_w1 := Burkert_OSCAT_BASIC.SCALE_R(X := Config.HLT.Assets.Level.EU, I_LO := 0.0, I_HI := Config.HLT.Assets.Level.Analog_Scale.Eu_Max, O_LO := 0, O_HI := 100);
Config.HLT.Current_Level_PCT := _w1;
Config.HLT.Current_Temp := Config.HLT.Assets.Temperature.EU;
_w2 := True;
IF _w2 THEN
    HLT_Task_Manager_0(Config := Config); // HLT_Task_Manager
END_IF
Service_Water_0(SFCReset := Config.HLT.Service_Water_Destination.eTarget <> Service_Water_0.Current_Destination, Config := Config); // Service_Water
IF Config.HLT.Mode.eMode=eHLT_Modes.Off THEN _w3 := False; END_IF
Config.HLT.AutoFill.Brew_Active := _w3;
_w4 := True;
IF _w4 THEN
    Alarm_Manager_0(Config := Config); // Alarm_Manager
END_IF
_w5 := _w4;
IF _w5 THEN
    HLT_Valve_Manager_0(Config := Config); // HLT_Valve_Manager
END_IF
_w6 := _w5;
IF _w6 THEN
    HLT_PID_Manager_0(Config := Config); // HLT_PID_MANAGER
END_IF
_w7 := _w6;
IF _w7 THEN
    HLT_Status_Manager_0(Config := Config); // HLT_STATUS_MANAGER
END_IF
IF _w7 THEN
    HLT_VFD_Ctrl_0(Config := Config); // HLT_VFD_Ctrl
END_IF
R_TRIG_1(CLK := Config.HLT.Mode.eMode<>HLT_Tasks_0.Current_Mode); // R_trig
IF _w2 THEN
    HLT_Tasks_0(SFCReset := R_TRIG_1.Q, Config := Config); // HLT_Tasks
END_IF
Config.HLT.Assets.Level.Burkert.cAlarm_Config := Config.HLT.AutoFill.Current_Profile.Level;
Config.HLT.Assets.Temperature.Burkert.cAlarm_Config := Config.HLT.AutoFill.Current_Profile.Temperature;
Config.HLT.Assets.HTX_Inlet_TT.Burkert.cAlarm_Config := Config.HLT.AutoFill.Current_Profile.Temperature;
Config.HLT.Assets.HTX_Outlet_TT.Burkert.cAlarm_Config := Config.HLT.AutoFill.Current_Profile.Temperature;
_w8 := DaySeconds(Hour := Config.HLT.Profile[1].Enable_Hour, Minute := Config.HLT.Profile[1].Enable_Minute, Second := 0);
_w9 := DaySeconds(Hour := Config.HLT.Profile[2].Enable_Hour, Minute := Config.HLT.Profile[2].Enable_Minute, Second := 0);
_w10 := DaySeconds(Hour := Config.HLT.Profile[3].Enable_Hour, Minute := Config.HLT.Profile[3].Enable_Minute, Second := 0);
_w11 := DaySeconds(Hour := Config.HLT.Profile[4].Enable_Hour, Minute := Config.HLT.Profile[4].Enable_Minute, Second := 0);
_w12 := Burkert_OSCAT_BASIC.BIT_OF_DWORD(in := Config.HLT.Profile[0].Enable_Days, N := RTC.wDayOfWeek);
_w13 := DaySeconds(Hour := Config.HLT.Profile[0].Enable_Hour, Minute := Config.HLT.Profile[0].Enable_Minute, Second := 0);
_w14 := (_w12 AND Day_Seconds = _w13 OR Config.HLT.AutoFill.Brew_Active) AND (Config	.HLT.Mode.eMode=eHLT_Modes.Auto) OR (Config.HLT.Manual_Profile=0);
_w15 := Burkert_OSCAT_BASIC.BIT_OF_DWORD(in := Config.HLT.Profile[1].Enable_Days, N := RTC.wDayOfWeek);
_w16 := _w15 AND Day_Seconds = _w8 AND (Config	.HLT.Mode.eMode=eHLT_Modes.Auto) OR (Config.HLT.Manual_Profile=1);
_w17 := Burkert_OSCAT_BASIC.BIT_OF_DWORD(in := Config.HLT.Profile[2].Enable_Days, N := RTC.wDayOfWeek);
_w18 := _w17 AND Day_Seconds = _w9 AND (Config	.HLT.Mode.eMode=eHLT_Modes.Auto) OR (Config.HLT.Manual_Profile=2);
_w19 := Burkert_OSCAT_BASIC.BIT_OF_DWORD(in := Config.HLT.Profile[3].Enable_Days, N := RTC.wDayOfWeek);
_w20 := _w19 AND Day_Seconds = _w10 OR (Config.HLT.Manual_Profile=3);
_w21 := Burkert_OSCAT_BASIC.BIT_OF_DWORD(in := Config.HLT.Profile[4].Enable_Days, N := RTC.wDayOfWeek);
_w22 := _w21 AND Day_Seconds = _w11 AND (Config	.HLT.Mode.eMode=eHLT_Modes.Auto) AND False OR (Config.HLT.Manual_Profile=4);
_w23 := _w14 OR _w16 OR _w18 OR _w20 OR _w22;
_w24 := SEL(_w14, SEL(_w16, SEL(_w18, SEL(_w20, SEL(_w22, 5, 4), 3), 2), 1), 0);
_w25 := _w23;
IF _w25 THEN _w26 := MUX(_w24, Config.HLT.Profile[0], Config.HLT.Profile[1], Config.HLT.Profile[2], Config.HLT.Profile[3], Config.HLT.Profile[4]); END_IF
Config.HLT.AutoFill.Current_Profile := _w26;
R_TRIG_2(CLK := _w25); // R_trig
IF R_TRIG_2.Q THEN _w27 := eHLT_Task.Fill; END_IF
Config.HLT.Task.eTask := _w27;
_w28 := _w23;
IF _w28 THEN _w29 := _w24; END_IF
Config.HLT.Active_Profile := _w29;
IF _w28 THEN _w30 := 255; END_IF
Config	.HLT.Manual_Profile := _w30;

END_PROGRAM

// HLT_Task_Manager
FUNCTION_BLOCK HLT_Task_Manager
VAR_INPUT
END_VAR
VAR_OUTPUT
END_VAR
VAR
END_VAR


VAR_INPUT
	Config: REFERENCE TO Config_DUT;
END_VAR
VAR // added by the converter: edge detectors and wires of the graphical bodies
    _w1 : BOOL;
END_VAR

_w1 := Config.HLT.AutoFill.Current_Profile.Temperature.Setpoints.Hi_warn - Config.HLT.AutoFill.Current_Profile.Temperature.Setpoints.Low_warn >= 2.0;
Config.HLT.Task.eTask := SEL(Config.HLT.Mode.eMode=eHlt_Modes.Auto, Config.HLT.Task.eTask, SEL(Config.HLT.Service_Water.OpenDestination, SEL(Config.HLT.Assets.Level.Status.eStatus=Burkert.eSensor_Status.Low_Low_Alarm, SEL(Config.HLT.Assets.Level.Status.eStatus=Burkert.eSensor_Status.Low_Warning, SEL(_w1 AND (Config.HLT.Assets.Temperature.EU < (Config.HLT.AutoFill.Current_Profile.Temperature.Setpoints.Low_warn+0.1)) OR (Config.HLT.Assets.Level.EU>(Config.HLT.Assets.Level.Burkert.cAlarm_Config.Hi_Warn-10)), SEL(_w1 AND (Config.HLT.Assets.Temperature.EU > (Config.HLT.AutoFill.Current_Profile.Temperature.Setpoints.Hi_warn-0.2)), SEL(NOT _w1 AND (Config.HLT.Assets.Temperature.EU > (Config.HLT.AutoFill.Current_Profile.Temperature.Setpoints.Low_warn)), Config.HLT.Task.eTask, eHLT_Task.Ready_Holding), eHLT_Task.Ready), eHLT_Task.Heat_Recirculate), eHLT_Task.Fill_Heat), eHLT_Task.Fill), eHLT_Task.Line_Chase));

END_FUNCTION_BLOCK

// Service_Water
FUNCTION_BLOCK Service_Water
VAR
	TransferLoop:Batch_Transfer;
	Current_Destination:INT;
	Current_Mode:INT;
	lclStatus:Transfer_Status;
END_VAR

VAR_INPUT
	SFCReset:BOOL;
	//Config.HLT.Service_Water.DestinationOpen:BOOL;
END_VAR

VAR_OUTPUT
	SFCcurrentStep:STRING[49];
	//Config.HLT.Service_Water.OpenDestination:BOOL;
END_VAR

VAR_IN_OUT
	//transfer:cBatch_Transfer;
END_VAR
VAR_INPUT
	Config: REFERENCE TO Config_DUT;
END_VAR

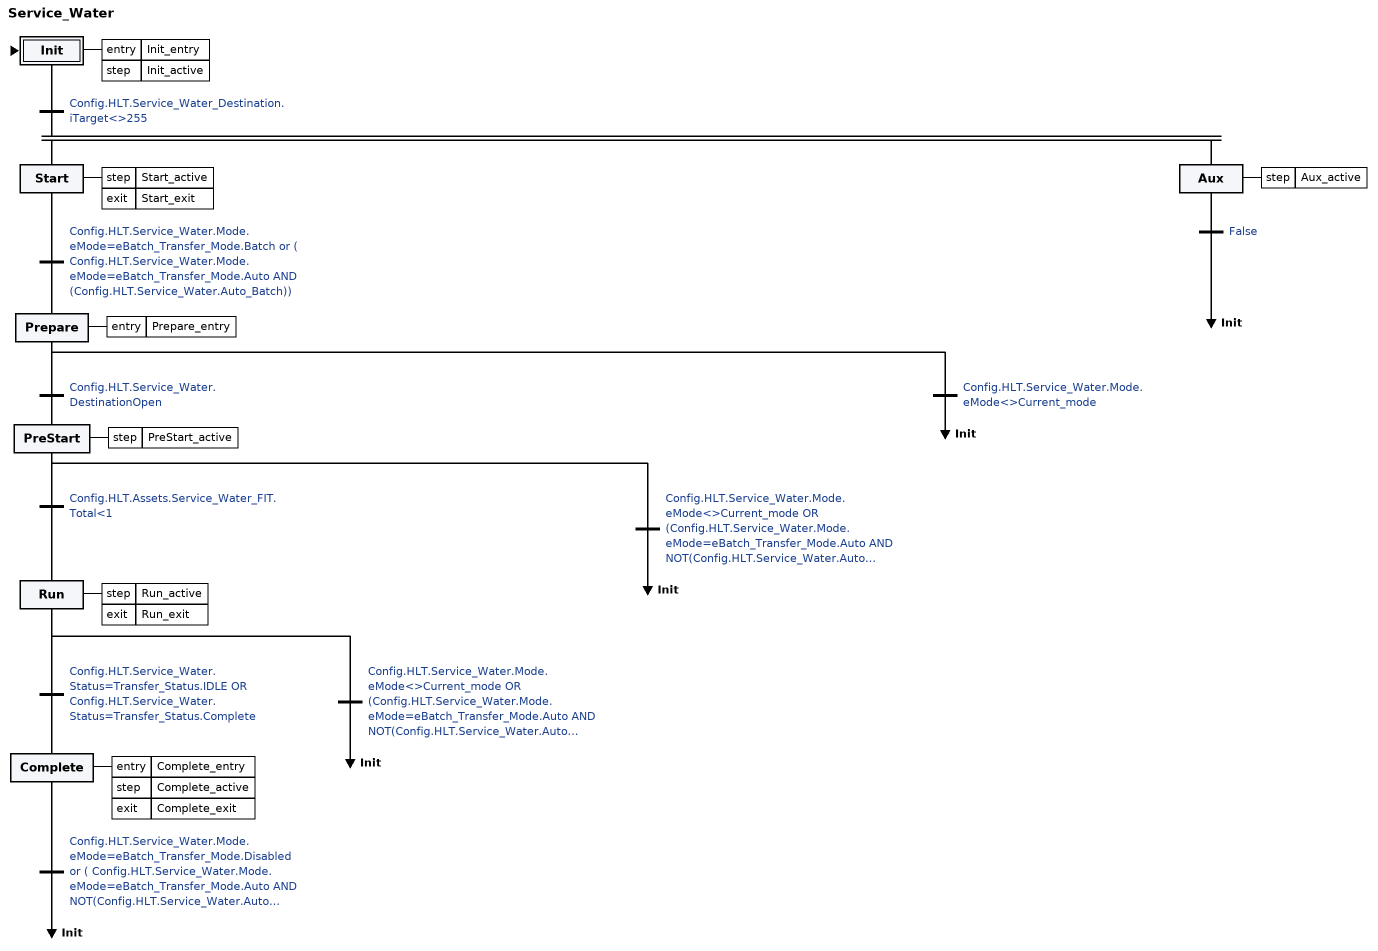
INITIAL_STEP Init:
    Init_entry(P1);  // entry action
    Init_active(N);  // step action
END_STEP
TRANSITION FROM Init TO (Start, Aux)
    := Config.HLT.Service_Water_Destination.iTarget<>255;
END_TRANSITION
STEP Start:
    Start_active(N);  // step action
    Start_exit(P0);  // exit action
END_STEP
STEP Aux:
    Aux_active(N);  // step action
END_STEP
TRANSITION FROM Aux TO Init
    := False;
END_TRANSITION
TRANSITION FROM Start TO Prepare
    := Config.HLT.Service_Water.Mode.eMode=eBatch_Transfer_Mode.Batch or ( Config.HLT.Service_Water.Mode.eMode=eBatch_Transfer_Mode.Auto AND (Config.HLT.Service_Water.Auto_Batch));
END_TRANSITION
STEP Prepare:
    Prepare_entry(P1);  // entry action
END_STEP
TRANSITION FROM Prepare TO PreStart
    := Config.HLT.Service_Water.DestinationOpen;
END_TRANSITION
TRANSITION FROM Prepare TO Init
    := Config.HLT.Service_Water.Mode.eMode<>Current_mode;
END_TRANSITION
STEP PreStart:
    PreStart_active(N);  // step action
END_STEP
TRANSITION FROM PreStart TO Run
    := Config.HLT.Assets.Service_Water_FIT.Total<1;
END_TRANSITION
TRANSITION FROM PreStart TO Init
    := Config.HLT.Service_Water.Mode.eMode<>Current_mode OR (Config.HLT.Service_Water.Mode.eMode=eBatch_Transfer_Mode.Auto AND NOT(Config.HLT.Service_Water.Auto_Batch));
END_TRANSITION
STEP Run:
    Run_active(N);  // step action
    Run_exit(P0);  // exit action
END_STEP
TRANSITION FROM Run TO Complete
    := Config.HLT.Service_Water.Status=Transfer_Status.IDLE OR Config.HLT.Service_Water.Status=Transfer_Status.Complete;
END_TRANSITION
TRANSITION FROM Run TO Init
    := Config.HLT.Service_Water.Mode.eMode<>Current_mode OR (Config.HLT.Service_Water.Mode.eMode=eBatch_Transfer_Mode.Auto AND NOT(Config.HLT.Service_Water.Auto_Batch));
END_TRANSITION
STEP Complete:
    Complete_entry(P1);  // entry action
    Complete_active(N);  // step action
    Complete_exit(P0);  // exit action
END_STEP
TRANSITION FROM Complete TO Init
    := Config.HLT.Service_Water.Mode.eMode=eBatch_Transfer_Mode.Disabled or ( Config.HLT.Service_Water.Mode.eMode=eBatch_Transfer_Mode.Auto AND NOT(Config.HLT.Service_Water.Auto_Batch));
END_TRANSITION

END_FUNCTION_BLOCK

// HLT_VFD_Ctrl
FUNCTION_BLOCK HLT_VFD_Ctrl
VAR
END_VAR
VAR_INPUT
	Config: REFERENCE TO Config_DUT;
END_VAR
VAR // added by the converter: edge detectors and wires of the graphical bodies
    _w1, _w2 : ANY;
END_VAR

_w1 := (Config.HLT.Assets.SprayBall.Status=Burkert.eBCV_Status.A_Open) AND (Config.HLT.Task.eTask=eHLT_Task.Spray_Ball);
Config.HLT.Assets.Mix_Pump.PLC_Run := (Config.HLT.Assets.Strike_HW.Valve_Actual>5) OR (Config.HLT.Assets.Sparge_HW.Valve_Actual>5) OR _w1;
Config.HLT.Assets.Mix_Pump.PLC_CMD := SEl(_w1, MAX(Config.HLT.Assets.Sparge_HW.Valve_Actual, Config.HLT.Assets.Strike_HW.Valve_Actual), Config.HLT.Spray_Ball_Rate);
_w2 := Config.HLT.Assets.PID_Recirc.CV + (Config	.HLT.Service_Water.ACV);
Config.HLT.Assets.Recirc_Pump.PLC_CMD := SEL(_w2 <= 15, LIMIT(0.0, 100.0, _w2), 15);
Config.HLT.Assets.Recirc_Pump.PLC_Run := 5 < _w2;
// Config.HLT.Assets.Sparge_CW.Valve_Actual>5: input not connected
// Config.HLT.Assets.Strike_HW.Valve_Actual>5: input not connected
// Config.HLT.Assets.PID_Recirc.CV>2: input not connected

END_FUNCTION_BLOCK

// HLT_Valve_Manager
FUNCTION_BLOCK HLT_Valve_Manager
VAR
	//TOF_0: TOF;
END_VAR
VAR_INPUT
	Config: REFERENCE TO Config_DUT;
END_VAR
VAR // added by the converter: edge detectors and wires of the graphical bodies
    _w1, _w2 : ANY;
END_VAR

_w1 := (Config.HLT.Task.eTask=eHLT_Task.Heat_Recirculate) OR (Config.HLT.Task.eTask=eHLT_Task.Fill) OR (Config.HLT.Task.eTask=eHLT_Task.Fill_Heat) OR (Config.HLT.Task.eTask=eHLT_Task.Ready) OR (Config.HLT.Task.eTask=eHLT_Task.Spray_Ball);
Config.HLT.Assets.HTX_Steam.PLC_CMD := MAX(Config.HLT.Assets.PID_HTX.CV, 0.0);
_w2 := NOT (Config.HLT.Mode.eMode=eHLT_Modes.Off) AND Config.HLT.Assets.Level.Ready AND (Config.HLT.Assets.Level.Status.eStatus<>Burkert.eSensor_Status.HiHi_Alarm) AND ((Config.HLT.Task.eTask=eHLT_Task.Fill) OR (Config.HLT.Task.eTask=eHLT_Task.Fill_Heat));
Config.HLT.Assets.CW_Fill.PLC_CMD := _w2;
Config.HLT.Assets.Recirc_To_HTX.PLC_CMD := _w1;
Config.HLT.Assets.HTX_Outlet_ACV.PLC_CMD := SEL(Config.HLT.Task.eTask=eHLT_Task.Line_Chase, SEL(_w2, SEL((Config.HLT.Task.eTask=eHLT_Task.Ready_Holding) OR (Config.HLT.Task.eTask=eHLT_Task.Heat_Recirculate) OR (Config.HLT.Task.eTask=eHLT_Task.Ready) OR Config.HLT.Assets.PID_Recirc.PLC_Enable, 0.0, Config.HLT.Assets.PID_Recirc.CV), 100), Config.HLT.Assets.PID_Recirc.CV);
Config.HLT.Assets.SprayBall.PLC_CMD := (Config.HLT.Task.eTask=eHLT_Task.Spray_Ball) OR False;

END_FUNCTION_BLOCK

// HLT_PID_Manager
FUNCTION_BLOCK HLT_PID_Manager
VAR 
	RAMP_REAL_0: RAMP_REAL;
END_VAR
VAR_INPUT
	Config: REFERENCE TO Config_DUT;
END_VAR


//Config.HLT.Assets.HTX_FIT
VAR // added by the converter: edge detectors and wires of the graphical bodies
    _w1, _w2, _w4 : BOOL;
    _w3, _w5 : ANY;
END_VAR

Config.HLT.Assets.PID_HTX.Actual := Config.HLT.Assets.HTX_Outlet_TT.EU;
Config.HLT.Assets.PID_Recirc.Actual := Config.HLT.Assets.HTX_FIT.Rate;
_w1 := (Config.HLT.Task.eTask=eHLT_Task.Line_Chase) OR (Config.HLT.Task.eTask=eHLT_Task.Heat_Recirculate) OR (Config.HLT.Task.eTask=eHLT_Task.Ready_Holding) OR False;
_w2 := ((Config.HLT.Task.eTask=eHLT_Task.Line_Chase) OR (Config.HLT.Task.eTask=eHLT_Task.Heat_Recirculate) OR (Config.HLT.Task.eTask=eHLT_Task.Ready_Holding) OR False OR (Config.HLT.Task.eTask=eHLT_Task.Heat_Recirculate) OR (Config.HLT.Task.eTask=eHLT_Task.Fill_Heat)) AND (Config.HLT.Assets.HTX_FIT.Rate>10);
IF _w2 THEN _w3 := SEL(Config.HLT.Task.eTask=eHLT_Task.Ready_Holding, Config.HLT.AutoFill.Current_Profile.Temperature.Setpoints.Hi_warn, Config.HLT.AutoFill.Current_Profile.Temperature.Setpoints.Low_warn + (Config.HLT.AutoFill.Current_Profile.Temperature.Setpoints.Hi_warn - Config.HLT.AutoFill.Current_Profile.Temperature.Setpoints.Low_warn) / 2.0); END_IF
Config.HLT.Assets.PID_HTX.PLC_Target := _w3;
Config.HLT.Assets.PID_HTX.PLC_Enable := _w2;
RAMP_REAL_0(
    IN := SEL(Config.HLT.Assets.PID_Recirc.CV>99, Config.HLT.recirc_Rate + Config.HLT.Service_Water.Config.Rate, Config.HLT.Service_Water.Config.Rate),
    ASCEND := 5,
    DESCEND := 1,
    TIMEBASE := T#2s,
    RESET := False); // RAMP_REAL
_w4 := _w1;
IF _w4 THEN _w5 := SEL(Config.HLT.Task.eTask=eHLT_Task.Line_Chase, Config.HLT.recirc_Rate, RAMP_REAL_0.OUT); END_IF
Config.HLT.Assets.PID_Recirc.PLC_Target := _w5;
Config.HLT.Assets.PID_Recirc.PLC_Enable := _w4;

END_FUNCTION_BLOCK

// HLT_Status_Manager
FUNCTION_BLOCK HLT_Status_Manager
VAR
	TON_0: TON;
END_VAR
VAR_INPUT
	Config: REFERENCE TO Config_DUT;
END_VAR

//Config.HLT.Assets.CW_Fill

(* body of a kind this reader does not render *)

END_FUNCTION_BLOCK

// Service_Water_Manager
FUNCTION_BLOCK Service_Water_Manager
VAR
	//tStr_Destination:Service_Water_mapping;
	Service_Water_0: Service_Water;
END_VAR

VAR_INPUT
	Config: REFERENCE TO Config_DUT;
END_VAR
VAR // added by the converter: edge detectors and wires of the graphical bodies
    _w1, _w2, _w3, _w4, _w5, _w6, _w7 : ANY;
END_VAR

_w1 := (Config.HLT.Service_Water_Destination.eTarget=Service_Water_mapping.MLT_Vessel) AND (Config.MM.Status=eMM_Status.Rinse_Vessel);
_w2 := (Config.HLT.Service_Water_Destination.eTarget=Service_Water_mapping.KTWP_Sprayball) AND (Config.KT.Status=eKT_Status.Rinse);
_w3 := (Config.HLT.Service_Water_Destination.eTarget=Service_Water_mapping.Grant_Chase) AND (Config.MM.Status=eMM_Status.Rinse_Grant) AND (GVL.BCV[BCV_Mapping.BCV_008_Drain_BCV].Status=Burkert.eBCV_Status.A_Open) AND (GVL.BCV[BCV_Mapping.BCV_010_Grant_Out].Status=Burkert.eBCV_Status.A_Open);
_w4 := (Config.HLT.Service_Water_Destination.eTarget=Service_Water_mapping.KTWP_Low_Outlet) AND (Config.KT.Status=eKT_Status.Rinse_Low_Outlet);
_w5 := (Config.HLT.Service_Water_Destination.eTarget=Service_Water_mapping.CastOut_Chase) AND ((Config.KT.Status=eKT_Status.CastOut_Chase_Start) OR (Config.KT.Status=eKT_Status.CastOut_Chase_Active));
_w6 := (Config.HLT.Service_Water_Destination.eTarget=Service_Water_mapping.KTWP_Sprayball) AND (Config.KT.Status=eKT_Status.Rinse_Tank);
_w7 := (Config.HLT.Service_Water_Destination.eTarget=Service_Water_mapping.MLT_Transfer_Chase) AND ((Config.MM.Status=eMM_Status.Transfer_Chase_Ready) OR (Config.MM.Status=eMM_Status.Transfer_Chase_Active));
Config.HLT.Service_Water.DestinationOpen := MUX(Config	.HLT	.Service_Water_Destination.iTarget, GVL.BCV[BCV_Mapping.Underlet].Status=Burkert.eBCV_Status.A_Open, GVL.BCV[BCV_Mapping.BCV_028_MLT_Line_Chase].Status=Burkert.eBCV_Status.A_Open, GVL.BCV[BCV_Mapping.BCV_031_Grant_Spray_Ball].Status=Burkert.eBCV_Status.A_Open, GVL.BCV[BCV_Mapping.BCV_001_KTWP_Service_water_in].Status=Burkert.eBCV_Status.A_Open, GVL.BCV[BCV_Mapping.BCV_029_rinse_valve ].Status=Burkert.eBCV_Status.A_Open, (GVL.BCV[BCV_Mapping.KTWP_Spray_Ball].Status=Burkert.eBCV_Status.A_Open) AND (GVL.BCV[BCV_Mapping.BCV_039].Status=Burkert.eBCV_Status.A_Open) AND (GVL.BCV[BCV_Mapping.BCV_001_KTWP_Service_water_in].Status=Burkert.eBCV_Status.A_Open), (GVL.BCV[BCV_Mapping.BCV_017_KTWP_Tangent_Recirc].Status=Burkert.eBCV_Status.A_Open) AND (GVL.BCV[BCV_Mapping.BCV_039].Status=Burkert.eBCV_Status.A_Open) AND (GVL.BCV[BCV_Mapping.BCV_001_KTWP_Service_water_in].Status=Burkert.eBCV_Status.A_Open), (GVL.BCV[BCV_Mapping.BCV_001_KTWP_Service_water_in].Status=Burkert.eBCV_Status.A_Open) AND (GVL.BCV[BCV_Mapping.BCV_023_KTWP_High_outlet].Status=Burkert.eBCV_Status.A_Open), (GVL.BCV[BCV_Mapping.BCV_001_KTWP_Service_water_in].Status=Burkert.eBCV_Status.A_Open) AND (GVL.BCV[BCV_Mapping.BCV_024_KTWP_Low_Outlet].Status=Burkert.eBCV_Status.A_Open), False);
Config.HLT.Service_Water.Auto_Batch := (Config.HLT.Service_Water.Mode.eMode=eBatch_Transfer_Mode.Auto) AND ((Config.HLT.Service_Water_Destination.eTarget=Service_Water_mapping.CastOut_Chase) AND (Config.KT.Status=eKT_Status.CastOut_Chase_Active) OR (Config.HLT.Service_Water_Destination.eTarget=Service_Water_mapping.MLT_UnderLet) AND ((Config.MM.Status=eMM_Status.Underlet_Start) OR (Config.MM.Status=eMM_Status.Underlet_Active) OR (Config.MM.Status=eMM_Status.Rinse_Underlet)) OR _w7 OR _w5 OR _w3 OR _w1 OR _w2 OR (Config.HLT.Service_Water_Destination.eTarget=Service_Water_mapping.KTWP_High_Outlet) AND (Config.KT.Status=eKT_Status.Rinse_High_Outlet) OR _w6 OR _w4);

END_FUNCTION_BLOCK

// HLT_Tasks_OLD
FUNCTION_BLOCK HLT_Tasks_OLD
VAR
	Current_Task:eHLT_Task;
	Current_Mode:eHLT_Modes;
END_VAR

VAR_INPUT
	SFCReset:BOOL;
	
END_VAR

VAR_OUTPUT
	SFCcurrentStep:STRING[49];
END_VAR
VAR_INPUT
	Config: REFERENCE TO Config_DUT;
END_VAR

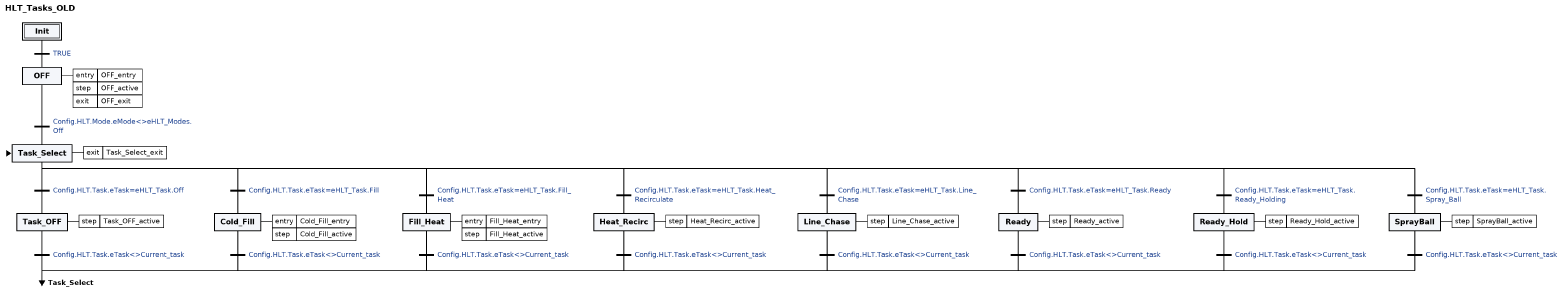
INITIAL_STEP Init:
END_STEP
TRANSITION FROM Init TO OFF
    := TRUE;
END_TRANSITION
STEP OFF:
    OFF_entry(P1);  // entry action
    OFF_active(N);  // step action
    OFF_exit(P0);  // exit action
END_STEP
TRANSITION FROM OFF TO Task_Select
    := Config.HLT.Mode.eMode<>eHLT_Modes.Off;
END_TRANSITION
STEP Task_Select:
    Task_Select_exit(P0);  // exit action
END_STEP
TRANSITION FROM Task_Select TO Task_OFF
    := Config.HLT.Task.eTask=eHLT_Task.Off;
END_TRANSITION
STEP Task_OFF:
    Task_OFF_active(N);  // step action
END_STEP
TRANSITION FROM Task_OFF TO Task_Select
    := Config.HLT.Task.eTask<>Current_task;
END_TRANSITION
TRANSITION FROM Task_Select TO Cold_Fill
    := Config.HLT.Task.eTask=eHLT_Task.Fill;
END_TRANSITION
STEP Cold_Fill:
    Cold_Fill_entry(P1);  // entry action
    Cold_Fill_active(N);  // step action
END_STEP
TRANSITION FROM Cold_Fill TO Task_Select
    := Config.HLT.Task.eTask<>Current_task;
END_TRANSITION
TRANSITION FROM Task_Select TO Fill_Heat
    := Config.HLT.Task.eTask=eHLT_Task.Fill_Heat;
END_TRANSITION
STEP Fill_Heat:
    Fill_Heat_entry(P1);  // entry action
    Fill_Heat_active(N);  // step action
END_STEP
TRANSITION FROM Fill_Heat TO Task_Select
    := Config.HLT.Task.eTask<>Current_task;
END_TRANSITION
TRANSITION FROM Task_Select TO Heat_Recirc
    := Config.HLT.Task.eTask=eHLT_Task.Heat_Recirculate;
END_TRANSITION
STEP Heat_Recirc:
    Heat_Recirc_active(N);  // step action
END_STEP
TRANSITION FROM Heat_Recirc TO Task_Select
    := Config.HLT.Task.eTask<>Current_task;
END_TRANSITION
TRANSITION FROM Task_Select TO Line_Chase
    := Config.HLT.Task.eTask=eHLT_Task.Line_Chase;
END_TRANSITION
STEP Line_Chase:
    Line_Chase_active(N);  // step action
END_STEP
TRANSITION FROM Line_Chase TO Task_Select
    := Config.HLT.Task.eTask<>Current_task;
END_TRANSITION
TRANSITION FROM Task_Select TO Ready
    := Config.HLT.Task.eTask=eHLT_Task.Ready;
END_TRANSITION
STEP Ready:
    Ready_active(N);  // step action
END_STEP
TRANSITION FROM Ready TO Task_Select
    := Config.HLT.Task.eTask<>Current_task;
END_TRANSITION
TRANSITION FROM Task_Select TO Ready_Hold
    := Config.HLT.Task.eTask=eHLT_Task.Ready_Holding;
END_TRANSITION
STEP Ready_Hold:
    Ready_Hold_active(N);  // step action
END_STEP
TRANSITION FROM Ready_Hold TO Task_Select
    := Config.HLT.Task.eTask<>Current_task;
END_TRANSITION
TRANSITION FROM Task_Select TO SprayBall
    := Config.HLT.Task.eTask=eHLT_Task.Spray_Ball;
END_TRANSITION
STEP SprayBall:
    SprayBall_active(N);  // step action
END_STEP
TRANSITION FROM SprayBall TO Task_Select
    := Config.HLT.Task.eTask<>Current_task;
END_TRANSITION

END_FUNCTION_BLOCK

// CIP_CTRL
PROGRAM CIP_CTRL
VAR
	R_TRIG_0: R_Trig;
	TON_0: TON;
	TON_1: TON;
	R_TRIG_1: R_Trig;
	TP_0: TP;
	TP_1: TP;
	TON_2: TON;
	Stage_Target_Out: REAL;
	Stage_Target_IN: REAL;
	TON_3: TON;
	F_TRIG_0: F_trig;
	Cip_Mode_tmp:eCIP_Modes;
	TP_2: TP;
	TP_3: TP;
	F_TRIG_1: F_trig;
	TON_4: TON;
	R_TRIG_2: R_trig;
	TP_4: TP;

	TON_3a: TON;
	TON_5: TON;
	TON_6: TON;
END_VAR
VAR // added by the converter: edge detectors and wires of the graphical bodies
    _w1, _w2, _w3, _w4, _w5, _w6, _w7, _w8, _w9, _w10, _w11, _w12, _w13, _w14, _w15, _w16, _w17, _w18, _w19, _w20, _w21, _w22, _w23 : BOOL;
    _rt1, _rt2, _rt3, _rt4, _rt5 : R_TRIG;
    _ft1 : F_TRIG;
END_VAR

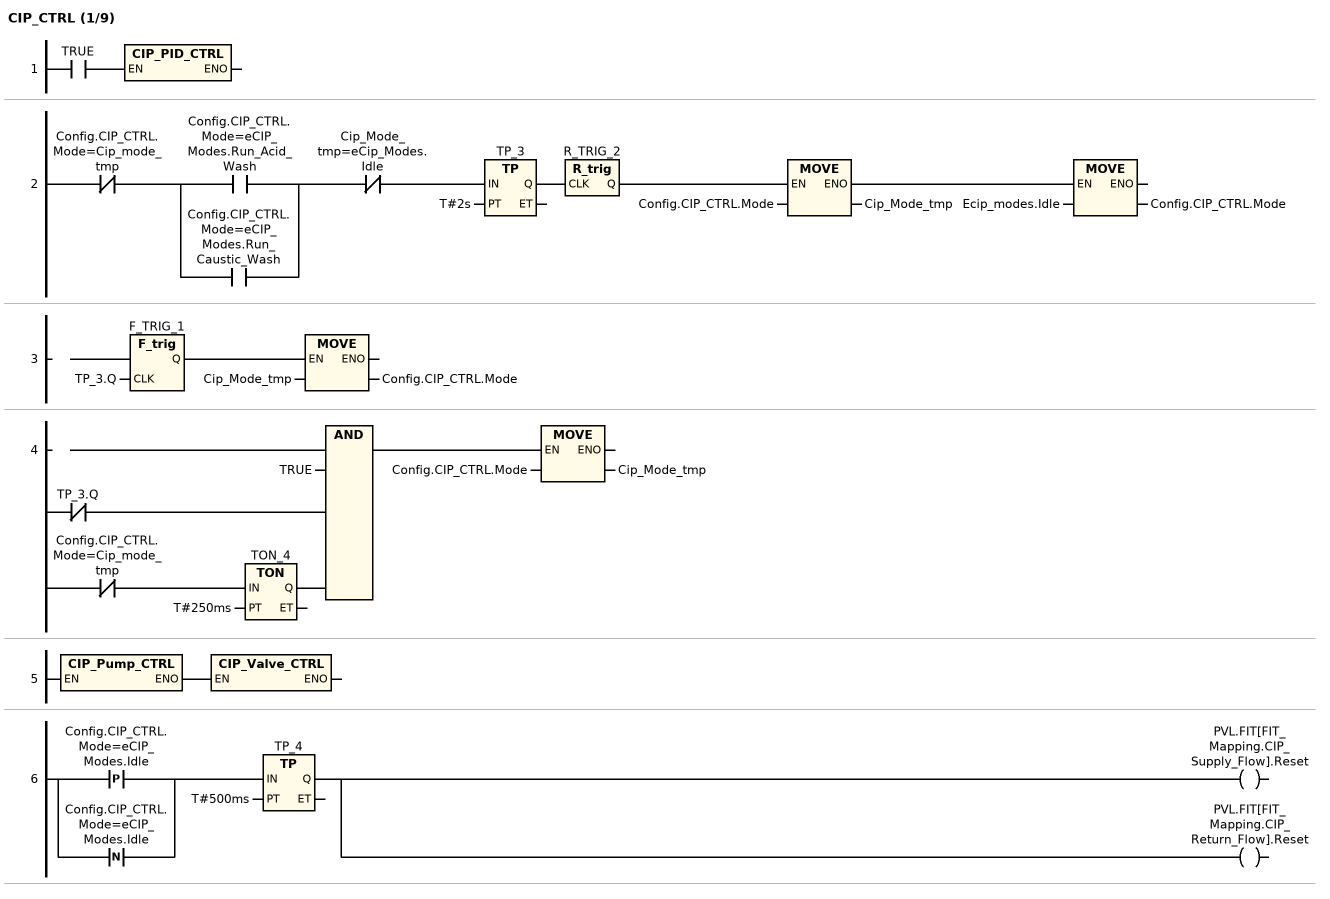
// NETWORK 1
CIP_PID_CTRL();

// NETWORK 2
TP_3(IN := NOT (Config.CIP_CTRL.Mode=Cip_mode_tmp) AND ((Config.CIP_CTRL.Mode=eCIP_Modes.Run_Acid_Wash) OR (Config.CIP_CTRL.Mode=eCIP_Modes.Run_Caustic_Wash)) AND NOT (Cip_Mode_tmp=eCip_Modes.Idle), PT := T#2s); // TP
R_TRIG_2(CLK := TP_3.Q); // R_trig
_w1 := R_TRIG_2.Q;
IF _w1 THEN Cip_Mode_tmp := Config.CIP_CTRL.Mode; END_IF
IF _w1 THEN Config.CIP_CTRL.Mode := Ecip_modes.Idle; END_IF

// NETWORK 3
F_TRIG_1(CLK := TP_3.Q); // F_trig
IF F_TRIG_1.Q THEN Config.CIP_CTRL.Mode := Cip_Mode_tmp; END_IF

// NETWORK 4
TON_4(IN := NOT (Config.CIP_CTRL.Mode=Cip_mode_tmp), PT := T#250ms); // TON
IF TRUE AND NOT TP_3.Q AND TON_4.Q THEN Cip_Mode_tmp := Config.CIP_CTRL.Mode; END_IF

// NETWORK 5
CIP_Pump_CTRL();
CIP_Valve_CTRL();

// NETWORK 6
_rt1(CLK := Config.CIP_CTRL.Mode=eCIP_Modes.Idle);
_ft1(CLK := Config.CIP_CTRL.Mode=eCIP_Modes.Idle);
TP_4(IN := _rt1.Q OR _ft1.Q, PT := T#500ms); // TP
PVL.FIT[FIT_Mapping.CIP_Supply_Flow].Reset := TP_4.Q;
PVL.FIT[FIT_Mapping.CIP_Return_Flow].Reset := TP_4.Q;

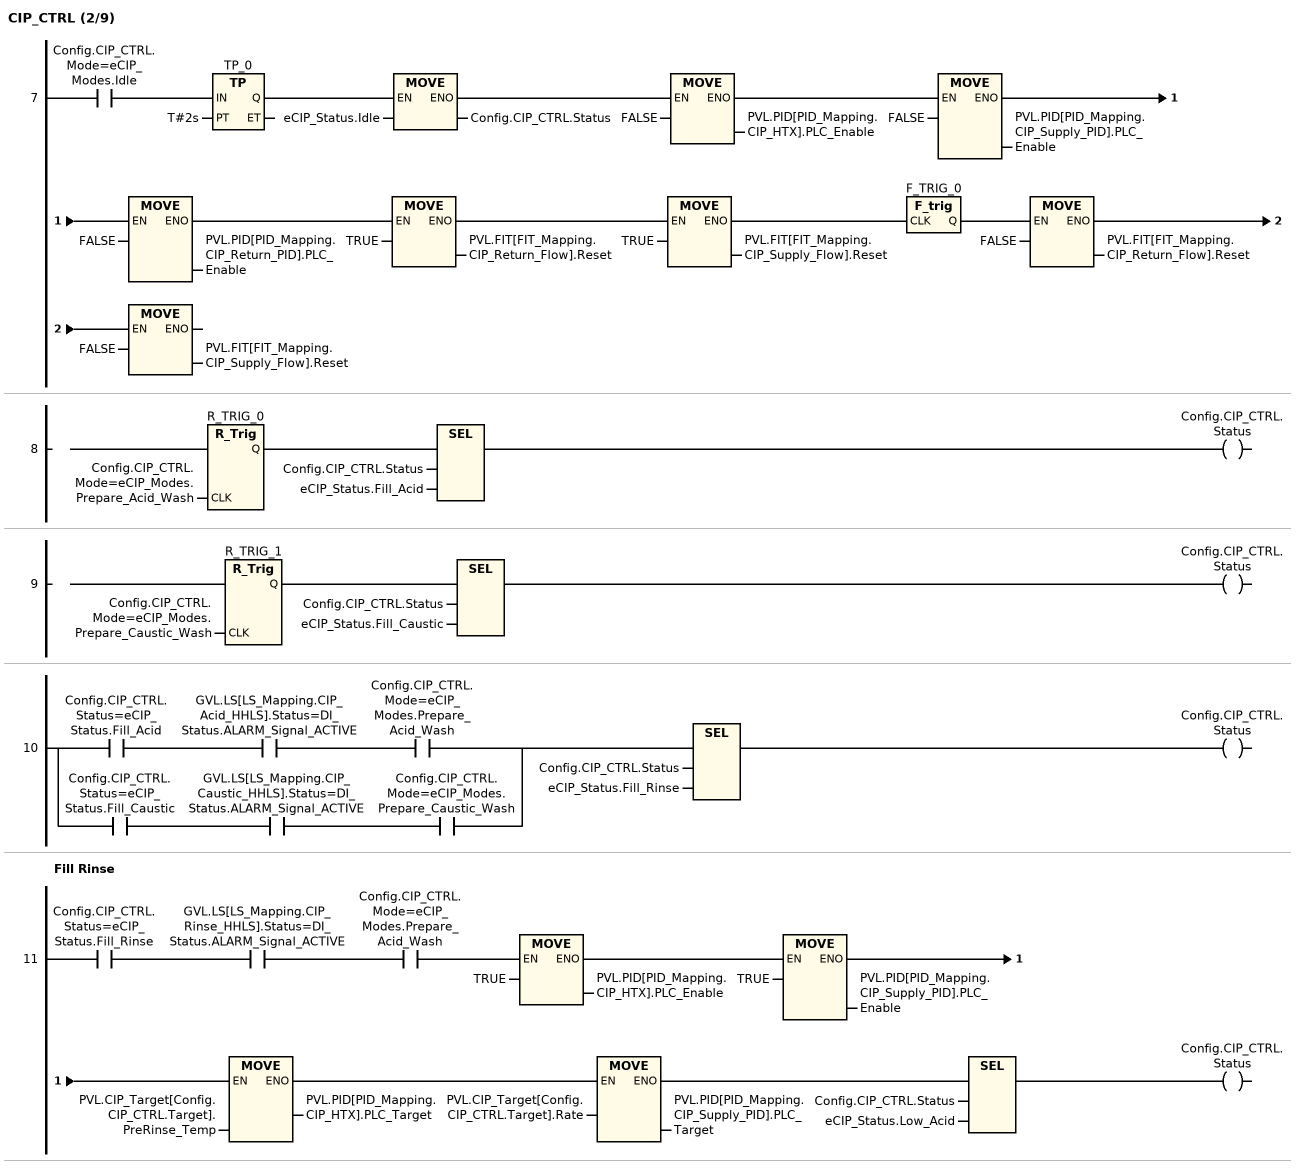
// NETWORK 7
TP_0(IN := Config.CIP_CTRL.Mode=eCIP_Modes.Idle, PT := T#2s); // TP
_w2 := TP_0.Q;
IF _w2 THEN Config.CIP_CTRL.Status := eCIP_Status.Idle; END_IF
IF _w2 THEN PVL.PID[PID_Mapping.CIP_HTX].PLC_Enable := FALSE; END_IF
IF _w2 THEN PVL.PID[PID_Mapping.CIP_Supply_PID].PLC_Enable := FALSE; END_IF
IF _w2 THEN PVL.PID[PID_Mapping.CIP_Return_PID].PLC_Enable := FALSE; END_IF
IF _w2 THEN PVL.FIT[FIT_Mapping.CIP_Return_Flow].Reset := TRUE; END_IF
IF _w2 THEN PVL.FIT[FIT_Mapping.CIP_Supply_Flow].Reset := TRUE; END_IF
F_TRIG_0(CLK := _w2); // F_trig
_w3 := F_TRIG_0.Q;
IF _w3 THEN PVL.FIT[FIT_Mapping.CIP_Return_Flow].Reset := FALSE; END_IF
IF _w3 THEN PVL.FIT[FIT_Mapping.CIP_Supply_Flow].Reset := FALSE; END_IF

// NETWORK 8
R_TRIG_0(CLK := Config.CIP_CTRL.Mode=eCIP_Modes.Prepare_Acid_Wash); // R_Trig
Config.CIP_CTRL.Status := SEL(R_TRIG_0.Q, Config.CIP_CTRL.Status, eCIP_Status.Fill_Acid);

// NETWORK 9
R_TRIG_1(CLK := Config.CIP_CTRL.Mode=eCIP_Modes.Prepare_Caustic_Wash); // R_Trig
Config.CIP_CTRL.Status := SEL(R_TRIG_1.Q, Config.CIP_CTRL.Status, eCIP_Status.Fill_Caustic);

// NETWORK 10
Config.CIP_CTRL.Status := SEL((Config.CIP_CTRL.Status=eCIP_Status.Fill_Acid) AND (GVL.LS[LS_Mapping.CIP_Acid_HHLS].Status=DI_Status.ALARM_Signal_ACTIVE) AND (Config.CIP_CTRL.Mode=eCIP_Modes.Prepare_Acid_Wash) OR (Config.CIP_CTRL.Status=eCIP_Status.Fill_Caustic) AND (GVL.LS[LS_Mapping.CIP_Caustic_HHLS].Status=DI_Status.ALARM_Signal_ACTIVE) AND (Config.CIP_CTRL.Mode=eCIP_Modes.Prepare_Caustic_Wash), Config.CIP_CTRL.Status, eCIP_Status.Fill_Rinse);

// NETWORK 11: Fill Rinse
_w4 := (Config.CIP_CTRL.Status=eCIP_Status.Fill_Rinse) AND (GVL.LS[LS_Mapping.CIP_Rinse_HHLS].Status=DI_Status.ALARM_Signal_ACTIVE) AND (Config.CIP_CTRL.Mode=eCIP_Modes.Prepare_Acid_Wash);
IF _w4 THEN PVL.PID[PID_Mapping.CIP_HTX].PLC_Enable := TRUE; END_IF
IF _w4 THEN PVL.PID[PID_Mapping.CIP_Supply_PID].PLC_Enable := TRUE; END_IF
IF _w4 THEN PVL.PID[PID_Mapping.CIP_HTX].PLC_Target := PVL.CIP_Target[Config.CIP_CTRL.Target].PreRinse_Temp; END_IF
IF _w4 THEN PVL.PID[PID_Mapping.CIP_Supply_PID].PLC_Target := PVL.CIP_Target[Config.CIP_CTRL.Target].Rate; END_IF
Config.CIP_CTRL.Status := SEL(_w4, Config.CIP_CTRL.Status, eCIP_Status.Low_Acid);

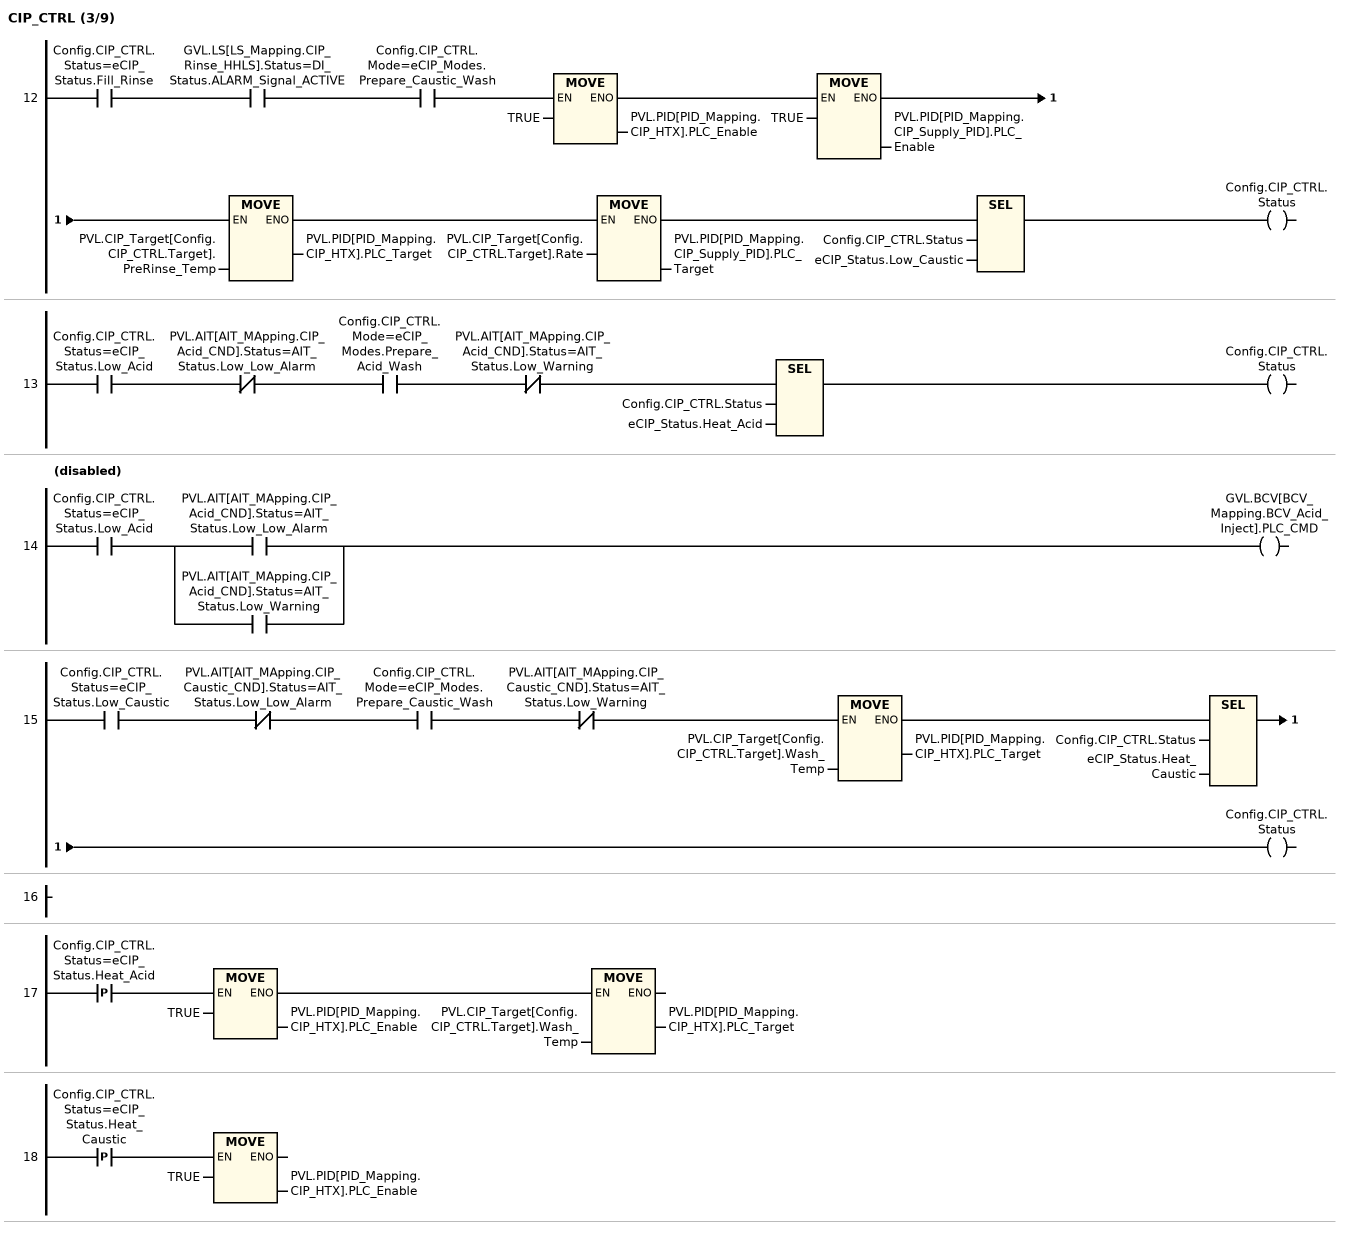
// NETWORK 12
_w5 := (Config.CIP_CTRL.Status=eCIP_Status.Fill_Rinse) AND (GVL.LS[LS_Mapping.CIP_Rinse_HHLS].Status=DI_Status.ALARM_Signal_ACTIVE) AND (Config.CIP_CTRL.Mode=eCIP_Modes.Prepare_Caustic_Wash);
IF _w5 THEN PVL.PID[PID_Mapping.CIP_HTX].PLC_Enable := TRUE; END_IF
IF _w5 THEN PVL.PID[PID_Mapping.CIP_Supply_PID].PLC_Enable := TRUE; END_IF
IF _w5 THEN PVL.PID[PID_Mapping.CIP_HTX].PLC_Target := PVL.CIP_Target[Config.CIP_CTRL.Target].PreRinse_Temp; END_IF
IF _w5 THEN PVL.PID[PID_Mapping.CIP_Supply_PID].PLC_Target := PVL.CIP_Target[Config.CIP_CTRL.Target].Rate; END_IF
Config.CIP_CTRL.Status := SEL(_w5, Config.CIP_CTRL.Status, eCIP_Status.Low_Caustic);

// NETWORK 13
Config.CIP_CTRL.Status := SEL((Config.CIP_CTRL.Status=eCIP_Status.Low_Acid) AND NOT (PVL.AIT[AIT_MApping.CIP_Acid_CND].Status=AIT_Status.Low_Low_Alarm) AND (Config.CIP_CTRL.Mode=eCIP_Modes.Prepare_Acid_Wash) AND NOT (PVL.AIT[AIT_MApping.CIP_Acid_CND].Status=AIT_Status.Low_Warning), Config.CIP_CTRL.Status, eCIP_Status.Heat_Acid);

// NETWORK 14 (disabled)
// GVL.BCV[BCV_Mapping.BCV_Acid_Inject].PLC_CMD := (Config.CIP_CTRL.Status=eCIP_Status.Low_Acid) AND ((PVL.AIT[AIT_MApping.CIP_Acid_CND].Status=AIT_Status.Low_Low_Alarm) OR (PVL.AIT[AIT_MApping.CIP_Acid_CND].Status=AIT_Status.Low_Warning));

// NETWORK 15
_w6 := (Config.CIP_CTRL.Status=eCIP_Status.Low_Caustic) AND NOT (PVL.AIT[AIT_MApping.CIP_Caustic_CND].Status=AIT_Status.Low_Low_Alarm) AND (Config.CIP_CTRL.Mode=eCIP_Modes.Prepare_Caustic_Wash) AND NOT (PVL.AIT[AIT_MApping.CIP_Caustic_CND].Status=AIT_Status.Low_Warning);
IF _w6 THEN PVL.PID[PID_Mapping.CIP_HTX].PLC_Target := PVL.CIP_Target[Config.CIP_CTRL.Target].Wash_Temp; END_IF
Config.CIP_CTRL.Status := SEL(_w6, Config.CIP_CTRL.Status, eCIP_Status.Heat_Caustic);

// NETWORK 16

// NETWORK 17
_rt2(CLK := Config.CIP_CTRL.Status=eCIP_Status.Heat_Acid);
_w7 := _rt2.Q;
IF _w7 THEN PVL.PID[PID_Mapping.CIP_HTX].PLC_Enable := TRUE; END_IF
IF _w7 THEN PVL.PID[PID_Mapping.CIP_HTX].PLC_Target := PVL.CIP_Target[Config.CIP_CTRL.Target].Wash_Temp; END_IF

// NETWORK 18
_rt3(CLK := Config.CIP_CTRL.Status=eCIP_Status.Heat_Caustic);
IF _rt3.Q THEN PVL.PID[PID_Mapping.CIP_HTX].PLC_Enable := TRUE; END_IF

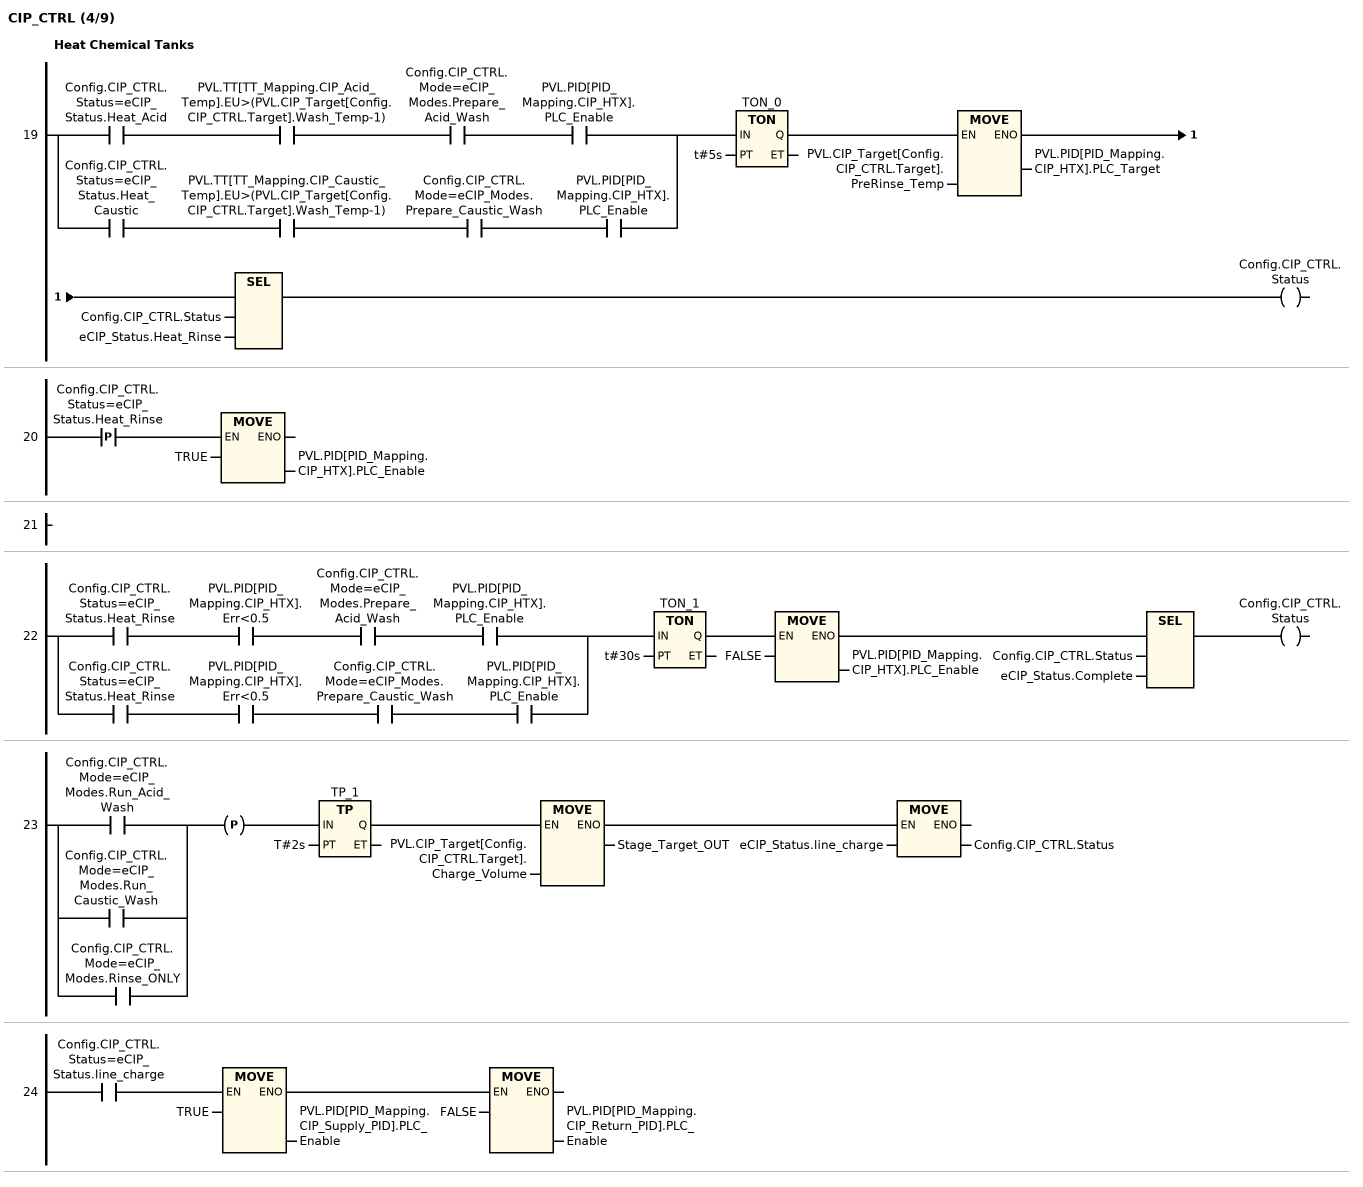
// NETWORK 19: Heat Chemical Tanks
TON_0(IN := (Config.CIP_CTRL.Status=eCIP_Status.Heat_Acid) AND (PVL.TT[TT_Mapping.CIP_Acid_Temp].EU>(PVL.CIP_Target[Config.CIP_CTRL.Target].Wash_Temp-1)) AND (Config.CIP_CTRL.Mode=eCIP_Modes.Prepare_Acid_Wash) AND PVL.PID[PID_Mapping.CIP_HTX].PLC_Enable OR (Config.CIP_CTRL.Status=eCIP_Status.Heat_Caustic) AND (PVL.TT[TT_Mapping.CIP_Caustic_Temp].EU>(PVL.CIP_Target[Config.CIP_CTRL.Target].Wash_Temp-1)) AND (Config.CIP_CTRL.Mode=eCIP_Modes.Prepare_Caustic_Wash) AND PVL.PID[PID_Mapping.CIP_HTX].PLC_Enable, PT := t#5s); // TON
_w8 := TON_0.Q;
IF _w8 THEN PVL.PID[PID_Mapping.CIP_HTX].PLC_Target := PVL.CIP_Target[Config.CIP_CTRL.Target].PreRinse_Temp; END_IF
Config.CIP_CTRL.Status := SEL(_w8, Config.CIP_CTRL.Status, eCIP_Status.Heat_Rinse);

// NETWORK 20
_rt4(CLK := Config.CIP_CTRL.Status=eCIP_Status.Heat_Rinse);
IF _rt4.Q THEN PVL.PID[PID_Mapping.CIP_HTX].PLC_Enable := TRUE; END_IF

// NETWORK 21

// NETWORK 22
TON_1(IN := (Config.CIP_CTRL.Status=eCIP_Status.Heat_Rinse) AND (PVL.PID[PID_Mapping.CIP_HTX].Err<0.5) AND (Config.CIP_CTRL.Mode=eCIP_Modes.Prepare_Acid_Wash) AND PVL.PID[PID_Mapping.CIP_HTX].PLC_Enable OR (Config.CIP_CTRL.Status=eCIP_Status.Heat_Rinse) AND (PVL.PID[PID_Mapping.CIP_HTX].Err<0.5) AND (Config.CIP_CTRL.Mode=eCIP_Modes.Prepare_Caustic_Wash) AND PVL.PID[PID_Mapping.CIP_HTX].PLC_Enable, PT := t#30s); // TON
_w9 := TON_1.Q;
IF _w9 THEN PVL.PID[PID_Mapping.CIP_HTX].PLC_Enable := FALSE; END_IF
Config.CIP_CTRL.Status := SEL(_w9, Config.CIP_CTRL.Status, eCIP_Status.Complete);

// NETWORK 23
_rt5(CLK := (Config.CIP_CTRL.Mode=eCIP_Modes.Run_Acid_Wash) OR (Config.CIP_CTRL.Mode=eCIP_Modes.Run_Caustic_Wash) OR (Config.CIP_CTRL.Mode=eCIP_Modes.Rinse_ONLY));
TP_1(IN := _rt5.Q, PT := T#2s); // TP
_w10 := TP_1.Q;
IF _w10 THEN Stage_Target_OUT := PVL.CIP_Target[Config.CIP_CTRL.Target].Charge_Volume; END_IF
IF _w10 THEN Config.CIP_CTRL.Status := eCIP_Status.line_charge; END_IF

// NETWORK 24
_w11 := Config.CIP_CTRL.Status=eCIP_Status.line_charge;
IF _w11 THEN PVL.PID[PID_Mapping.CIP_Supply_PID].PLC_Enable := TRUE; END_IF
IF _w11 THEN PVL.PID[PID_Mapping.CIP_Return_PID].PLC_Enable := FALSE; END_IF

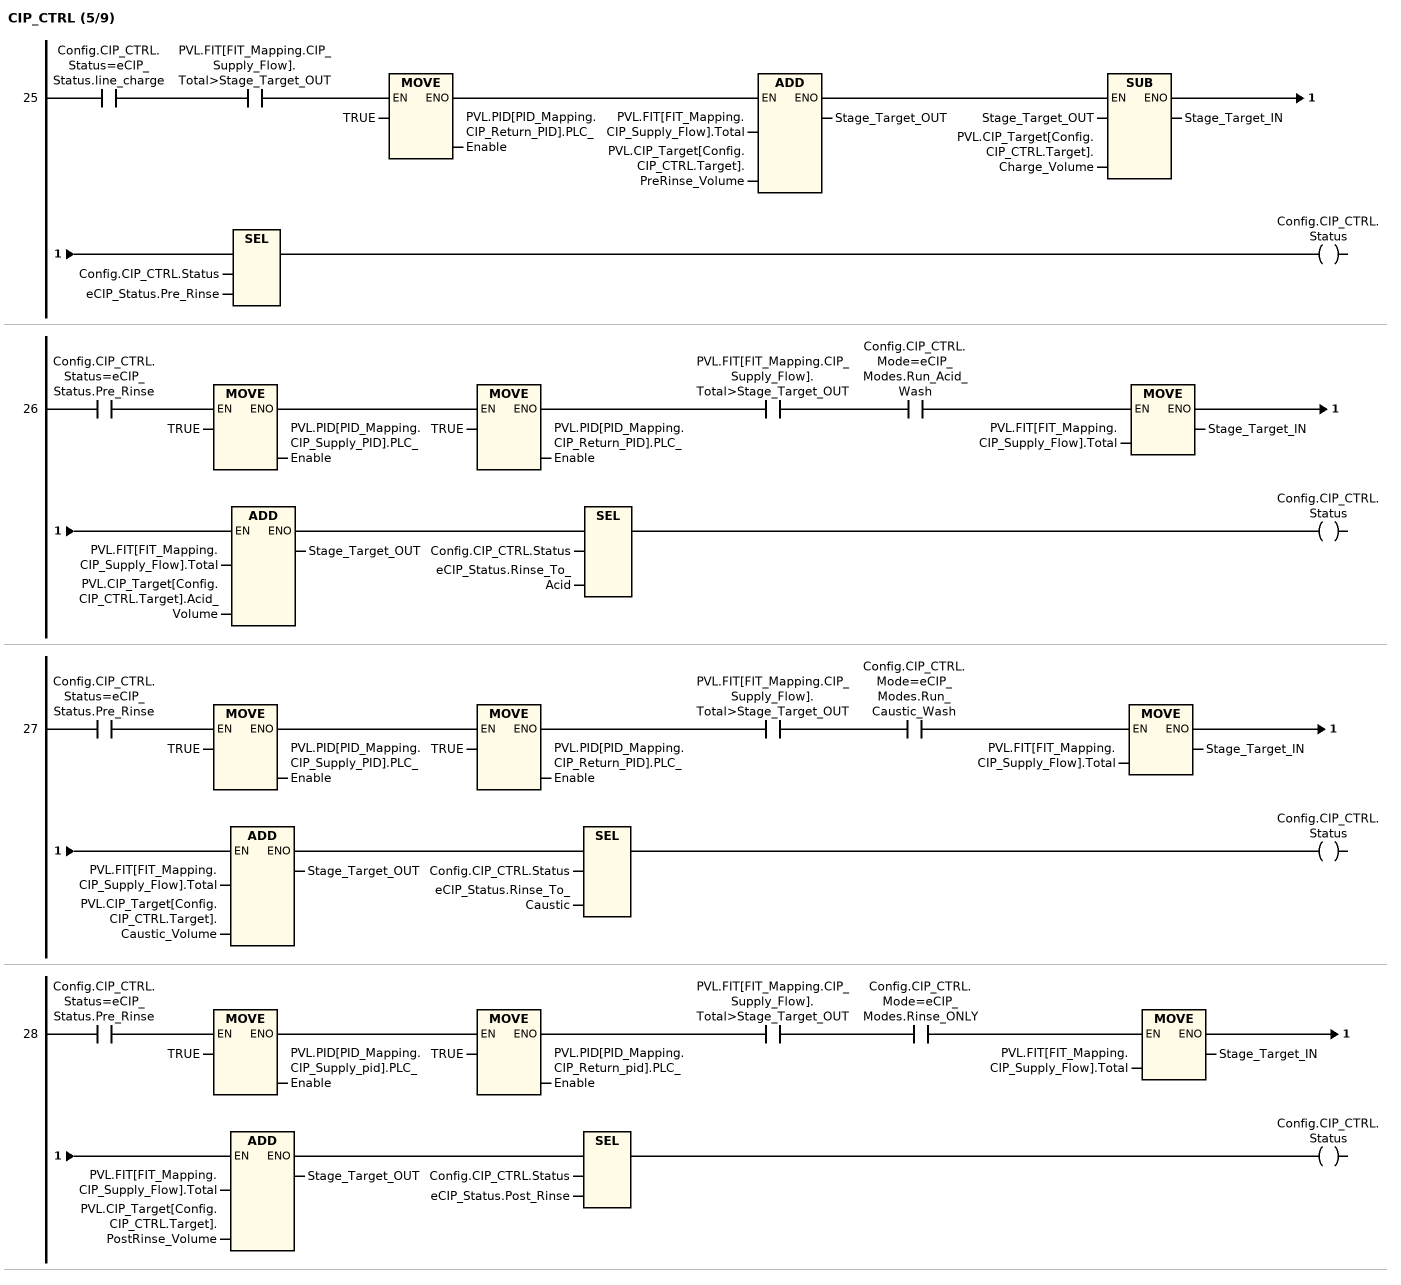
// NETWORK 25
_w12 := (Config.CIP_CTRL.Status=eCIP_Status.line_charge) AND (PVL.FIT[FIT_Mapping.CIP_Supply_Flow].Total>Stage_Target_OUT);
IF _w12 THEN PVL.PID[PID_Mapping.CIP_Return_PID].PLC_Enable := TRUE; END_IF
IF _w12 THEN
    Stage_Target_OUT := PVL.FIT[FIT_Mapping.CIP_Supply_Flow].Total + PVL.CIP_Target[Config.CIP_CTRL.Target].PreRinse_Volume;
END_IF
IF _w12 THEN Stage_Target_IN := Stage_Target_OUT - PVL.CIP_Target[Config.CIP_CTRL.Target].Charge_Volume; END_IF
Config.CIP_CTRL.Status := SEL(_w12, Config.CIP_CTRL.Status, eCIP_Status.Pre_Rinse);

// NETWORK 26
_w13 := Config.CIP_CTRL.Status=eCIP_Status.Pre_Rinse;
IF _w13 THEN PVL.PID[PID_Mapping.CIP_Supply_PID].PLC_Enable := TRUE; END_IF
IF _w13 THEN PVL.PID[PID_Mapping.CIP_Return_PID].PLC_Enable := TRUE; END_IF
IF _w13 AND (PVL.FIT[FIT_Mapping.CIP_Supply_Flow].Total>Stage_Target_OUT) AND (Config.CIP_CTRL.Mode=eCIP_Modes.Run_Acid_Wash) THEN
    Stage_Target_IN := PVL.FIT[FIT_Mapping.CIP_Supply_Flow].Total;
END_IF
IF _w13 AND (PVL.FIT[FIT_Mapping.CIP_Supply_Flow].Total>Stage_Target_OUT) AND (Config.CIP_CTRL.Mode=eCIP_Modes.Run_Acid_Wash) THEN
    Stage_Target_OUT := PVL.FIT[FIT_Mapping.CIP_Supply_Flow].Total + PVL.CIP_Target[Config.CIP_CTRL.Target].Acid_Volume;
END_IF
Config.CIP_CTRL.Status := SEL(_w13 AND (PVL.FIT[FIT_Mapping.CIP_Supply_Flow].Total>Stage_Target_OUT) AND (Config.CIP_CTRL.Mode=eCIP_Modes.Run_Acid_Wash), Config.CIP_CTRL.Status, eCIP_Status.Rinse_To_Acid);

// NETWORK 27
_w14 := Config.CIP_CTRL.Status=eCIP_Status.Pre_Rinse;
IF _w14 THEN PVL.PID[PID_Mapping.CIP_Supply_PID].PLC_Enable := TRUE; END_IF
IF _w14 THEN PVL.PID[PID_Mapping.CIP_Return_PID].PLC_Enable := TRUE; END_IF
IF _w14 AND (PVL.FIT[FIT_Mapping.CIP_Supply_Flow].Total>Stage_Target_OUT) AND (Config.CIP_CTRL.Mode=eCIP_Modes.Run_Caustic_Wash) THEN
    Stage_Target_IN := PVL.FIT[FIT_Mapping.CIP_Supply_Flow].Total;
END_IF
IF _w14 AND (PVL.FIT[FIT_Mapping.CIP_Supply_Flow].Total>Stage_Target_OUT) AND (Config.CIP_CTRL.Mode=eCIP_Modes.Run_Caustic_Wash) THEN
    Stage_Target_OUT := PVL.FIT[FIT_Mapping.CIP_Supply_Flow].Total + PVL.CIP_Target[Config.CIP_CTRL.Target].Caustic_Volume;
END_IF
Config.CIP_CTRL.Status := SEL(_w14 AND (PVL.FIT[FIT_Mapping.CIP_Supply_Flow].Total>Stage_Target_OUT) AND (Config.CIP_CTRL.Mode=eCIP_Modes.Run_Caustic_Wash), Config.CIP_CTRL.Status, eCIP_Status.Rinse_To_Caustic);

// NETWORK 28
_w15 := Config.CIP_CTRL.Status=eCIP_Status.Pre_Rinse;
IF _w15 THEN PVL.PID[PID_Mapping.CIP_Supply_pid].PLC_Enable := TRUE; END_IF
IF _w15 THEN PVL.PID[PID_Mapping.CIP_Return_pid].PLC_Enable := TRUE; END_IF
IF _w15 AND (PVL.FIT[FIT_Mapping.CIP_Supply_Flow].Total>Stage_Target_OUT) AND (Config.CIP_CTRL.Mode=eCIP_Modes.Rinse_ONLY) THEN
    Stage_Target_IN := PVL.FIT[FIT_Mapping.CIP_Supply_Flow].Total;
END_IF
IF _w15 AND (PVL.FIT[FIT_Mapping.CIP_Supply_Flow].Total>Stage_Target_OUT) AND (Config.CIP_CTRL.Mode=eCIP_Modes.Rinse_ONLY) THEN
    Stage_Target_OUT := PVL.FIT[FIT_Mapping.CIP_Supply_Flow].Total + PVL.CIP_Target[Config.CIP_CTRL.Target].PostRinse_Volume;
END_IF
Config.CIP_CTRL.Status := SEL(_w15 AND (PVL.FIT[FIT_Mapping.CIP_Supply_Flow].Total>Stage_Target_OUT) AND (Config.CIP_CTRL.Mode=eCIP_Modes.Rinse_ONLY), Config.CIP_CTRL.Status, eCIP_Status.Post_Rinse);

